{attribute 'qualified_only'}
TYPE E_SensirionFMMode :
(
	OK          := 0,
	OverRange   := 1,
	UnderRange  := 2,
	FlowInvalid := 3
);
END_TYPE

(* stored: Version 1.1.0.1, ProductVersion 3.1.4024.2
   EnumerationTextList E_SensirionFMMode: Id {b98576dc-259c-4b6c-8290-2e89870ef292} *)
